(* CoDeSys 2.3 export: SETMUOUTPUT.EXP *)

(* POU New Folder/setMUOutput, ST *)
FUNCTION setMUOutput : REAL
VAR_INPUT
	IN : BOOL;
END_VAR
VAR
END_VAR
IF IN THEN
	setMUOutput := 1.0;
ELSE
	setMUOutput := 0.0;
END_IF;
END_FUNCTION
